FUNCTION_BLOCK ILOCK_T_FF_AX (* Composite FB for a lockable toggle flip-flop with AE2 adapter interface, AX Out *)
  (* Standard: 61499-2; Description: Copyright (c) 2023 HR Agrartechnik GmbH This program and the accompanying materials are made available under the terms of the Eclipse Public License 2.0 which is available at https://www.eclipse.org/legal/epl-2.0/ SPDX-License-Identifier: EPL-2.0 *)
  (* Version 1.0, 2026-04-19, Franz Höpfinger, HR Agrartechnik GmbH, initial API and implementation and/or initial documentation *)
  PACKAGE logiBUS::signalprocessing::interlock;
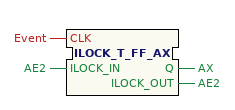
  EVENT_INPUT
    CLK; (* Clock for triggering a output toggle *)
  END_EVENT
  SOCKETS
    ILOCK_IN : adapter::types::bidirectional::AE2;
  END_SOCKETS
  PLUGS
    Q : adapter::types::unidirectional::AX; (* Output *)
    ILOCK_OUT : adapter::types::bidirectional::AE2;
  END_PLUGS
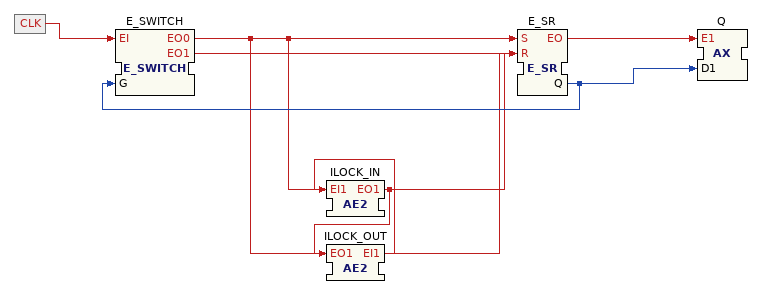
  FBS
    E_SR : iec61499::events::E_SR;
    E_SWITCH : iec61499::events::E_SWITCH;
  END_FBS
  EVENT_CONNECTIONS
    E_SWITCH.EO0 TO E_SR.S;
    E_SWITCH.EO1 TO E_SR.R;
    E_SWITCH.EO0 TO ILOCK_OUT.EO1;
    ILOCK_IN.EO1 TO E_SR.R;
    ILOCK_OUT.EI1 TO E_SR.R;
    E_SWITCH.EO0 TO ILOCK_IN.EI1;
    E_SR.EO TO Q.E1;
    CLK TO E_SWITCH.EI;
    ILOCK_IN.EO1 TO ILOCK_OUT.EO1;
    ILOCK_OUT.EI1 TO ILOCK_IN.EI1;
  END_CONNECTIONS
  DATA_CONNECTIONS
    E_SR.Q TO E_SWITCH.G;
    E_SR.Q TO Q.D1;
  END_CONNECTIONS
END_FUNCTION_BLOCK
